// TIA Portal V16 export
// export: Created 2022-09-01T14:29:21.5668028Z, ExportSetting WithDefaults, DisplayName Totally Integrated Automation Portal, DisplayVersion V16, DisplayName TIA Portal Version Control Interface, DisplayVersion V16, DisplayName TIA Portal Openness, DisplayVersion V16, DisplayName STEP 7 Professional, DisplayVersion V16, DisplayName STEP 7 Safety, DisplayVersion V16, DisplayName WinCC Advanced, DisplayVersion V16
DATA_BLOCK "Etapas_Grafcet_3"   // DB3
{ S7_Optimized_Access := 'TRUE' }
VERSION : 0.1
// stored: AutoNumber true, IsOnlyStoredInLoadMemory false, IsRetainMemResEnabled false, IsWriteProtectedInAS false, MemoryReserve 100
   VAR RETAIN
      ETAPA_13 : Bool;
      ETAPA_14 : Bool;
      ETAPA_15 : Bool;
      RESET_ETAPA_13 : Bool;
   END_VAR
BEGIN
END_DATA_BLOCK
